Fanuc TP program (LS listing): f7on.ls

/PROG  F7ON
/ATTR
OWNER		= MNEDITOR;
COMMENT		= "";
PROG_SIZE	= 120;
CREATE		= DATE 18-03-12  TIME 09:27:28;
MODIFIED	= DATE 18-03-12  TIME 09:29:18;
FILE_NAME	= ;
VERSION		= 0;
LINE_COUNT	= 1;
MEMORY_SIZE	= 460;
PROTECT		= READ_WRITE;
TCD:  STACK_SIZE	= 0,
      TASK_PRIORITY	= 50,
      TIME_SLICE	= 0,
      BUSY_LAMP_OFF	= 0,
      ABORT_REQUEST	= 0,
      PAUSE_REQUEST	= 0;
DEFAULT_GROUP	= *,*,*,*,*,*,*;
CONTROL_CODE	= 00000000 00000000;
/MN
   1:  F[7]=(ON) ;
/POS
/END
